Fanuc KAREL source: VT_READ_PQ.kl

PROGRAM T
%NOLOCKGROUP
VAR
 v0 : INTEGER
 v1 : PATH
 v2 : INTEGER
BEGIN
 VT_READ_PQ(v0, v1, v2)
END T
